FUNCTION TryConvert_LINT_TO_USINT : BOOL
VAR_INPUT
	in : LINT;
	out : REFERENCE TO USINT;
END_VAR

IF in > DatatypeLimits.MAX_VALUE_OF_LINT_WHICH_CAN_BE_HELD_IN_A_USINT THEN
	RETURN;
END_IF

IF in < DatatypeLimits.MIN_VALUE_OF_LINT_WHICH_CAN_BE_HELD_IN_A_USINT THEN
	RETURN;
END_IF

out := LINT_TO_USINT(in);
TryConvert_LINT_TO_USINT := TRUE;

END_FUNCTION

(* stored: Version 1.1.0.1, ProductVersion 3.1.4024.12
   POU TryConvert_LINT_TO_USINT: Id {cf30f086-de4e-4b3c-936e-633aea1dfde5}, SpecialFunc None *)
